PROGRAM pouS6Alarms
VAR
	idbMsgAlarm: FB_CheckMessageBounds;

END_VAR

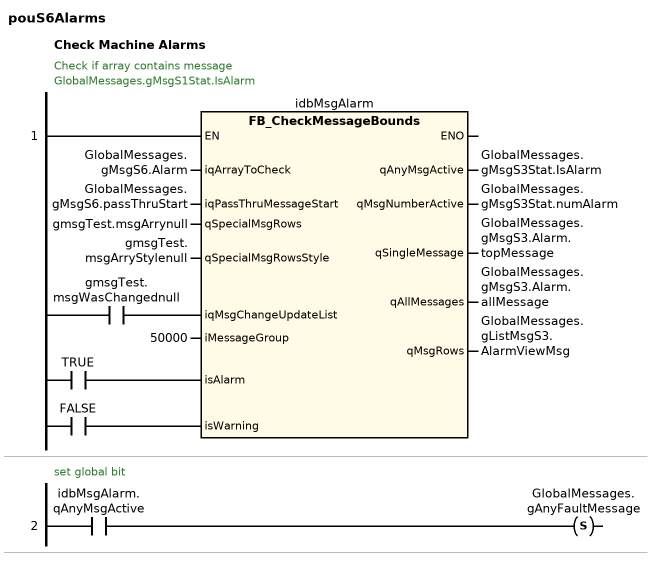
// NETWORK 1: Check Machine Alarms
// Check if array contains message
//
// GlobalMessages.gMsgS1Stat.IsAlarm
idbMsgAlarm(
    iqArrayToCheck := GlobalMessages.gMsgS6.Alarm,
    iqPassThruMessageStart := GlobalMessages.gMsgS6.passThruStart,
    qSpecialMsgRows := gmsgTest.msgArrynull,
    qSpecialMsgRowsStyle := gmsgTest.msgArryStylenull,
    iqMsgChangeUpdateList := gmsgTest.msgWasChangednull,
    iMessageGroup := 50000,
    isAlarm := TRUE,
    isWarning := FALSE,
    qAnyMsgActive => GlobalMessages.gMsgS3Stat.IsAlarm,
    qMsgNumberActive => GlobalMessages.gMsgS3Stat.numAlarm,
    qSingleMessage => GlobalMessages.gMsgS3.Alarm.topMessage,
    qAllMessages => GlobalMessages.gMsgS3.Alarm.allMessage,
    qMsgRows => GlobalMessages.gListMsgS3.AlarmViewMsg); // FB_CheckMessageBounds

// NETWORK 2
// set global bit
GlobalMessages.gAnyFaultMessage S= idbMsgAlarm.qAnyMsgActive;

END_PROGRAM

(* stored: Version 1.1.0.1, ProductVersion 3.1.4024.12
   POU pouS6Alarms: Id {eb79deb6-216d-4dca-ab86-2d4bfd70047a}, SpecialFunc None *)
